RESOURCE_TYPE _Core1
  (* Standard: 61499-2 *)
  (* Version 0.1, 2017-00-09, hpea485, UOA *)
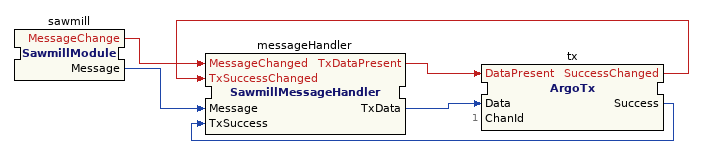
  FBS
    sawmill : SawmillModule;
    messageHandler : SawmillMessageHandler;
    tx : ArgoTx(ChanId := 1);
  END_FBS
  EVENT_CONNECTIONS
    sawmill.MessageChange TO messageHandler.MessageChanged;
    messageHandler.TxDataPresent TO tx.DataPresent;
    tx.SuccessChanged TO messageHandler.TxSuccessChanged;
  END_CONNECTIONS
  DATA_CONNECTIONS
    sawmill.Message TO messageHandler.Message;
    messageHandler.TxData TO tx.Data;
    tx.Success TO messageHandler.TxSuccess;
  END_CONNECTIONS
END_RESOURCE_TYPE
